// TIA Portal V20 export
FUNCTION_BLOCK "LConSMC_OverspeedDetection"   // FB86, SCL
TITLE = Enable Template
AUTHOR : (department/personInCharge/contact)
FAMILY : (family)
VERSION : 0.0.0.0
// Template for an FB with Enable / Valid handling based on PLCopen standard "Function Blocks for Motion Control" V2.0
// stored: Access Published, IsIECCheckEnabled true, MemoryReserve 100, SetENOAutomatically true
   VAR_INPUT
      enable { ExternalAccessible := 'False'; ExternalVisible := 'False'; ExternalWritable := 'False'} : Bool;   // TRUE: Enable functionality of FB
      reset { ExternalAccessible := 'False'; ExternalVisible := 'False'; ExternalWritable := 'False'} : Bool;   // TRUE: Reset preControlAdjust to 1.0 after a runaway detection
      vLine { ExternalAccessible := 'False'; ExternalVisible := 'False'; ExternalWritable := 'False'} : LReal;   // [m/min]/[ft/min] Line velocity setpoint
      vOverride { ExternalAccessible := 'False'; ExternalVisible := 'False'; ExternalWritable := 'False'} : LReal;   // [m/min]/[ft/min] Velocity override value (Correct sign required)
      vAct { ExternalAccessible := 'False'; ExternalVisible := 'False'; ExternalWritable := 'False'} : LReal;   // [m/min]/[ft/min] Actual circumference velocity of drive
      velocityDeviationLimit { ExternalAccessible := 'False'; ExternalVisible := 'False'; ExternalWritable := 'False'} : LReal := 10.0;   // [%] Maximum velocity deviation to detect drive runaway. Value is a percentage value of the entered vOverride.
      tCycle { ExternalAccessible := 'False'; ExternalVisible := 'False'; ExternalWritable := 'False'} : Real := 0.0;   // [ms] Cycle time the function block is called
   END_VAR
   VAR_OUTPUT
      valid { ExternalAccessible := 'False'; ExternalVisible := 'False'; ExternalWritable := 'False'} : Bool;   // TRUE: Valid set of output values available at the FB
      busy { ExternalAccessible := 'False'; ExternalVisible := 'False'; ExternalWritable := 'False'} : Bool;   // TRUE: FB is not finished and new output values can be expected
      error { ExternalAccessible := 'False'; ExternalVisible := 'False'; ExternalWritable := 'False'} : Bool;   // TRUE: An error occurred during the execution of the FB
      status { ExternalAccessible := 'False'; ExternalVisible := 'False'; ExternalWritable := 'False'} : Word;   // 16#0000 - 16#7FFF: Status of the FB, 16#8000 - 16#FFFF: Error identification
      effectiveLimit { ExternalAccessible := 'False'; ExternalVisible := 'False'; ExternalWritable := 'False'} : LReal;   // [m/min]/[ft/min] Maximum deviation before a runaway is detected
      runAway { ExternalAccessible := 'False'; ExternalVisible := 'False'; ExternalWritable := 'False'} : Bool;   // TRUE: The velocity deviation is too high, a runaway has been detected and the adjustment factor is ramped to 0.0
      preControlAdjust { ExternalAccessible := 'False'; ExternalVisible := 'False'; ExternalWritable := 'False'} : LReal := 1.0;   // [0..1] Adjustment factor for-pre control if a runaway has been detected
   END_VAR
   VAR
      statEnableOld { ExternalAccessible := 'False'; ExternalVisible := 'False'; ExternalWritable := 'False'} : Bool;   // Old value of 'enable' input for edge detection
      statValid { ExternalAccessible := 'False'; ExternalVisible := 'False'; ExternalWritable := 'False'} : Bool;   // Static value for output 'valid'
      statBusy { ExternalAccessible := 'False'; ExternalVisible := 'False'; ExternalWritable := 'False'} : Bool;   // Static value for output 'busy'
      statError { ExternalAccessible := 'False'; ExternalVisible := 'False'; ExternalWritable := 'False'} : Bool;   // Static value for output 'error'
      statErrorUserCleared { ExternalAccessible := 'False'; ExternalVisible := 'False'; ExternalWritable := 'False'} : Bool;   // Error occurred that can only be solved by user; rising edge at enable input necessary
      statErrorAutoCleared { ExternalAccessible := 'False'; ExternalVisible := 'False'; ExternalWritable := 'False'} : Bool;   // Error occurred that can be acknowledged by FB
      statStatus { ExternalAccessible := 'False'; ExternalVisible := 'False'; ExternalWritable := 'False'} : Word;   // Static value for output 'status'
      statFBState { ExternalAccessible := 'False'; ExternalVisible := 'False'; ExternalWritable := 'False'} : DInt;   // State in the state machine of the FB
      statDisablingCompleted { ExternalAccessible := 'False'; ExternalVisible := 'False'; ExternalWritable := 'False'} : Bool;   // TRUE: Disabling has been completed
      statABSvDiff { ExternalAccessible := 'False'; ExternalVisible := 'False'; ExternalWritable := 'False'} : LReal;   // [m/min]/[ft/min] Velocity deviation between setpoint and actual value
      statvDiffAdjustment { ExternalAccessible := 'False'; ExternalVisible := 'False'; ExternalWritable := 'False'} : LReal;
      statPrecontrolAdjust { ExternalAccessible := 'False'; ExternalVisible := 'False'; ExternalWritable := 'False'} : LReal := 1.0;
      instPT1 { ExternalAccessible := 'False'; ExternalVisible := 'False'; ExternalWritable := 'False'} : "LConSMC_PT1";
      statRunAwayDetected { ExternalAccessible := 'False'; ExternalVisible := 'False'; ExternalWritable := 'False'} : Bool;   // TRUE: An overspeed has been detected
      statResetOld { ExternalAccessible := 'False'; ExternalVisible := 'False'; ExternalWritable := 'False'} : Bool;
   END_VAR
   VAR_TEMP
      tempEnable : Bool;   // Temporary value for input 'enable'
      tempRunAwayLimit : LReal;
   END_VAR
   VAR CONSTANT
      SMOOTHING_TIME : Real := 100.0;   // [ms] PT1 time to ramp down scaling factor for torque precontrol
      FB_STATE_NO_PROCESSING : DInt := 0;   // FB state: No processing
      FB_STATE_ENABLING : DInt := 10;   // FB state: Enabling
      FB_STATE_PROCESSING : DInt := 50;   // FB state: Processing
      FB_STATE_DISABLING : DInt := 90;   // FB state: Disabling
      STATUS_NO_CALL : Word := 16#7000;   // No job being currently processed
      STATUS_FIRST_CALL : Word := 16#7001;   // First call after incoming new job (rising edge 'enable')
      STATUS_SUBSEQUENT_CALL : Word := 16#7002;   // Subsequent call during active processing without further details
      ERR_UNDEFINED_STATE : Word := 16#8600;
   END_VAR
BEGIN
   REGION BLOCK INFO HEADER
     //===============================================================================
     // SIEMENS AG / (c)Copyright 2023
     //-------------------------------------------------------------------------------
     // Title:            LConSMC_OverspeedDetection
     // Comment/Function: This function block detects a drive overspeed in torque controlled modes
     // Library/Family:   LConSMC
     // Author:           APC Erlangen
     // Tested with:      FW 2.8
     // Engineering:      TIA Portal V16
     // Restrictions:     -
     // Requirements:     -
     //-------------------------------------------------------------------------------
     // Change log table:
     // Version  | Date       | Expert in charge       | Changes applied
     //----------|------------|------------------------|------------------------------
     // 01.00.00 | 2023-11-07 | APC Erlangen           | Creation
     //===============================================================================
   END_REGION BLOCK INFO HEADER

   REGION DESCRIPTION
   (/*This function blocks monitors the deviation between line velocity setpoint and actual circumference velocity of the drive.
   If the deviation is bigger as the configured limit (vOverride + velocityDeviationLimit/100 * vOverride) the output "preControlAdjust" is ramped to 0.0 to
   disable the torque pre-control.*/)
   END_REGION DESCRIPTION

   #tempEnable := #enable; // Work with temporary value / create process image

   REGION ENABLING/DISABLING
     IF (#tempEnable = TRUE) AND (#statStatus = #STATUS_NO_CALL) THEN // Enable FB
       // First call; initialize FB
       #statValid := TRUE;
       #statBusy := TRUE;
       #statError := FALSE;
       #statStatus := #STATUS_FIRST_CALL;
       #statErrorUserCleared := FALSE;
       #statErrorAutoCleared := FALSE;
       #statDisablingCompleted := FALSE;
       // State machine - start functionality
       #statFBState := #FB_STATE_ENABLING;

       #statvDiffAdjustment := 1.0;
       #statPrecontrolAdjust := 1.0;
       #statRunAwayDetected := FALSE;
     ELSIF (#tempEnable = FALSE) AND (#statEnableOld = TRUE) THEN // Disable FB 
       #statFBState := #FB_STATE_DISABLING;

     ELSIF (#statStatus = #STATUS_FIRST_CALL) THEN // Set status identifier of subsequent call
       #statStatus := #STATUS_SUBSEQUENT_CALL;
     END_IF;

     // Edge detection 'enable' input
     #statEnableOld := #tempEnable;
   END_REGION ENABLING/DISABLING

   IF (#statStatus = #STATUS_NO_CALL) THEN // Nothing to do -> End here to reduce "system load"
     RETURN;
   END_IF;

   REGION STATE MACHINE
     CASE #statFBState OF // State machine of FB
       #FB_STATE_NO_PROCESSING:
         REGION No Processing
           // No processing active (Note: this state must always be present and left empty)
           ;
         END_REGION No Processing

       #FB_STATE_ENABLING: // Enabling active
         REGION enabling
           #statvDiffAdjustment := 1.0 + ABS(#velocityDeviationLimit)/100.0;
           #statFBState := #FB_STATE_PROCESSING;

         END_REGION enabling

       #FB_STATE_PROCESSING: // Processing active
         REGION Processing
           #tempRunAwayLimit := ABS(#vOverride) * #statvDiffAdjustment;
           #statABSvDiff := ABS((#vLine + #vOverride) - #vAct);

           IF #statABSvDiff > #tempRunAwayLimit THEN
             #statRunAwayDetected := TRUE;
           ELSIF #reset AND NOT #statResetOld THEN
             #statRunAwayDetected := FALSE;
           END_IF;

           #instPT1(set           := NOT #statRunAwayDetected,
                    x             := 0.0,
                    setvalue      := 1.0,
                    smoothingTime := #SMOOTHING_TIME,
                    tCycle        := #tCycle);

           #statPrecontrolAdjust := LIMIT(MN := 0.0,IN := #instPT1.y,MX := 1.0);

         END_REGION Processing

       #FB_STATE_DISABLING: // Disabling active
         REGION Disabling
           // When disabling is complete the bit #statDisablingCompleted must be set

           #statDisablingCompleted := TRUE;
         END_REGION Disabling

       ELSE // Undefined state in state machine reached
         REGION Undefined state
           #statStatus := #ERR_UNDEFINED_STATE;
           #statErrorUserCleared := TRUE;
         END_REGION Undefined state
     END_CASE;
     #statResetOld := #reset;
   END_REGION STATE MACHINE

   REGION OUTPUTS
     // Write outputs
     IF (#statDisablingCompleted = TRUE) THEN
       REGION Disabling
         // Reset outputs if disabling completed
         #statValid := FALSE;
         #statBusy := FALSE;
         #statError := FALSE;
         #statErrorUserCleared := FALSE;
         #statErrorAutoCleared := FALSE;
         #statStatus := #STATUS_NO_CALL;
         // TODO: Reset application specific outputs
         #statPrecontrolAdjust := 1.0;
         #statRunAwayDetected := FALSE;
       END_REGION Disabling

     ELSIF (#statErrorUserCleared = TRUE) AND (#statError = FALSE) THEN
       REGION Error user cleared
         // Error can only be cleared by user; rising edge at enable input is needed to continue 
         #statValid := FALSE;
         #statBusy := FALSE;
         #statError := TRUE;
         // execution aborted --> set state no processing
         #statFBState := #FB_STATE_NO_PROCESSING;
       END_REGION Error user cleared

     ELSIF (#statErrorAutoCleared = TRUE) AND (#statError = FALSE) THEN
       REGION Error auto cleared
         // Error can be reset by FB automatically  
         #statValid := FALSE;
         #statBusy := TRUE;
         #statError := TRUE;
         // TODO: Handling of autocleared error
         // 
       END_REGION Error auto cleared

     ELSIF (#statErrorAutoCleared = FALSE) AND (#statErrorUserCleared = FALSE) AND (#statError = TRUE) THEN
       REGION After user/auto cleared
         // If autocleared error is acknowledged
         #statValid := TRUE;
         #statBusy := TRUE;
         #statError := FALSE;
         // TODO: remove this line if more detailed status information is used instead of "#STATUS_SUBSEQUENT_CALL"
         #statStatus := #STATUS_SUBSEQUENT_CALL;
       END_REGION After user/auto cleared
     END_IF;

     REGION Write static values to outputs
       // Write static values to outputs
       #valid := #statValid;
       #busy := #statBusy;
       #error := #statError;
       #status := #statStatus;
       // if ENO mechanism is not used / not wanted replace the following line by --> ENO := TRUE;
       ENO := NOT #statError;
       // TODO: Write application specific static values to outputs
       #preControlAdjust := #statPrecontrolAdjust;
       #runAway := #statRunAwayDetected;
       #effectiveLimit := #tempRunAwayLimit;
     END_REGION Write static values to outputs
   END_REGION OUTPUTS
END_FUNCTION_BLOCK
